PROGRAM MAIN
VAR
END_VAR

END_PROGRAM

(* stored: Version 1.1.0.1
   POU MAIN: Id {77b06159-e118-453f-b4ba-28db65f215f2} *)
